INTERFACE EventLogger

METHOD save
VAR_INPUT
  execute: BOOL;
  data_ptr: PVOID;
  data_size: DWORD;
END_VAR
END_METHOD

END_INTERFACE

(* stored: Version 1.1.0.1, ProductVersion 3.1.4022.18
   Itf EventLogger: Id {ed02ee8e-c48d-425b-b1ba-db2fe412fd83}
   Method save: Id {bf8cf63d-c744-4436-8e81-8bfe67c7f6c9} *)
